(* IEC 61131-3 sources: 2026_Projet_YGO_ExcavatriceDragage/CODE/TESTS, 3 files *)

(* ---- PRG_SafetyValidation.st ---- *)
(* ═══════════════════════════════════════════════════════════════
   🧪 PRG_SafetyValidation — Validateur Automatique de Sécurité (CI/CD)
   ───────────────────────────────────────────────────────────────
   🎯 Rôle : Exécute une suite de scénarios de tests réglementaires
      (NF EN ISO 13849-1) sur le bloc FB_Safety_EmergencyManagement.
   ⚙️ S'exécute uniquement si GVL_Simulation.SimulationModeActive est actif.
   ═══════════════════════════════════════════════════════════════ *)

PROGRAM PRG_SafetyValidation
VAR_OUTPUT
    // Rapport de test (CI/CD)
    TestInProgress             : BOOL;
    TC01_NominalArming_Ok      : BOOL;
    TC02_RedundancyFault_Ok    : BOOL;
    TC03_Lockout_Ok            : BOOL;
    AllTestsPassed             : BOOL;
    TestFailed                 : BOOL;
    FailedTestCase             : INT;         // Numéro du scénario en échec
END_VAR
VAR
    StartTests                 : BOOL;        // Commande de démarrage des tests
    TestSeqStep                : INT := 0;    // Séquenceur de test
    TestTimer                  : TON;         // Timer d'attente d'étapes
    OverrideChainTrue          : BOOL := FALSE; // Force l'entrée boucle d'urgence à TRUE
    OverrideChainFalse         : BOOL := FALSE; // Force l'entrée boucle d'urgence à FALSE
    OverrideContactorFalse     : BOOL := FALSE; // Force l'entrée contacteur à FALSE

    // Signaux locaux pour stimuler le bloc sous test
    ArmRequest                 : BOOL;
    ResetFaults                : BOOL;
    CmdEmergencyCutOff         : BOOL;
END_VAR

// === IMPLEMENTATION ===

// ⛔ Neutralisation si la simulation globale n'est pas active (sécurité physique)
IF NOT GVL_Simulation.SimulationModeActive THEN
    TestSeqStep := 0;
    TestInProgress := FALSE;
    RETURN;
END_IF;

// ⏱️ Timer général d'étape
TestTimer(IN := (TestSeqStep <> 0), PT := T#10s);

// 🔀 Séquenceur de Test Automatique
CASE TestSeqStep OF

    0: // IDLE — En attente du départ de test
        IF StartTests THEN
            StartTests := FALSE;
            TestInProgress := TRUE;
            TC01_NominalArming_Ok := FALSE;
            TC02_RedundancyFault_Ok := FALSE;
            TC03_Lockout_Ok := FALSE;
            AllTestsPassed := FALSE;
            TestFailed := FALSE;
            FailedTestCase := 0;
            OverrideChainTrue := FALSE;
            OverrideChainFalse := FALSE;
            OverrideContactorFalse := FALSE;
            TestSeqStep := 10;
        END_IF;

    // ─────────────────────────────────────────────────────────────────
    // 🧪 SCÉNARIO 1 : Séquence Nominale (TC-01)
    // ─────────────────────────────────────────────────────────────────
    10: // Phase 1.1 : Initialisation saine
        ResetFaults := TRUE;
        IF NOT PRG_10_Outputs.instSafetyEmergencyManagement.RedundancyTestFailed AND
           NOT PRG_10_Outputs.instSafetyEmergencyManagement.EmergencyArmingFailed THEN
            ResetFaults := FALSE;
            TestSeqStep := 11;
        END_IF;

    11: // Phase 1.2 : Envoi demande réarmement
        ArmRequest := TRUE;
        TestSeqStep := 12;

    12: // Phase 1.3 : Vérification début d'auto-test
        ArmRequest := FALSE;
        IF PRG_10_Outputs.instSafetyEmergencyManagement.ArmingSeqStep = 1 THEN
            TestSeqStep := 13;
        END_IF;

    13: // Phase 1.4 : Attente réussite de l'auto-test et début impulsion armement
        IF PRG_10_Outputs.instSafetyEmergencyManagement.ArmingSeqStep = 5 THEN
            TestSeqStep := 14;
        END_IF;

    14: // Phase 1.5 : Attente fin de l'impulsion et confirmation armement
        IF PRG_00_Inputs.EmergencyStopOk AND PRG_10_Outputs.instSafetyEmergencyManagement.ArmingSeqStep = 0 THEN
            // Armé nominalement ! Maintenant on teste le Trip d'urgence
            TestSeqStep := 15;
        END_IF;

    15: // Phase 1.6 : Simulation d'un appui bouton d'urgence (Coupure franche)
        OverrideChainFalse := TRUE;
        TestSeqStep := 16;

    16: // Phase 1.7 : Vérification coupure instantanée
        IF NOT PRG_10_Outputs.PowerCutOff_A_RQ AND NOT PRG_10_Outputs.PowerCutOff_B_RQ AND NOT PRG_00_Inputs.EmergencyStopOk THEN
            // Coupure validée, on relâche le bouton d'urgence (doit rester coupé)
            OverrideChainFalse := FALSE;
            TestSeqStep := 17;
        END_IF;

    17: // Phase 1.8 : Vérification de l'auto-maintien (Latch)
        IF NOT PRG_10_Outputs.PowerCutOff_A_RQ AND NOT PRG_10_Outputs.PowerCutOff_B_RQ THEN
            TC01_NominalArming_Ok := TRUE;
            TestSeqStep := 20; // Passer au test de redondance
        ELSE
            TestFailed := TRUE;
            FailedTestCase := 1;
            TestSeqStep := 999;
        END_IF;

    // ─────────────────────────────────────────────────────────────────
    // 🧪 SCÉNARIO 2 : Défaut de Redondance (TC-02)
    // ─────────────────────────────────────────────────────────────────
    20: // Phase 2.1 : Acquitter le défaut précédent et relancer l'armement
        ResetFaults := TRUE;
        IF NOT PRG_10_Outputs.instSafetyEmergencyManagement.RedundancyTestFailed THEN
            ResetFaults := FALSE;
            ArmRequest := TRUE;
            TestSeqStep := 21;
        END_IF;

    21: // Phase 2.2 : Attente de l'auto-test canal A
        ArmRequest := FALSE;
        IF PRG_10_Outputs.instSafetyEmergencyManagement.ArmingSeqStep = 1 THEN
            // Simuler contacteur A soudé : la chaîne d'urgence reste fermée (TRUE)
            // malgré l'ordre de coupure du canal A.
            OverrideChainTrue := TRUE;
            TestSeqStep := 22;
        END_IF;

    22: // Phase 2.3 : Vérification de la détection du défaut (dans les 200ms)
        IF PRG_10_Outputs.instSafetyEmergencyManagement.RedundancyTestFailed AND
           PRG_10_Outputs.instSafetyEmergencyManagement.ArmingSeqStep = 0 THEN
            // Détection réussie ! Les sorties doivent être inhibées.
            OverrideChainTrue := FALSE;
            TC02_RedundancyFault_Ok := TRUE;
            TestSeqStep := 30; // Passer au test de Lockout
        ELSIF TestTimer.Q THEN
            // Timeout -> Échec du test de redondance
            OverrideChainTrue := FALSE;
            TestFailed := TRUE;
            FailedTestCase := 2;
            TestSeqStep := 999;
        END_IF;

    // ─────────────────────────────────────────────────────────────────
    // 🧪 SCÉNARIO 3 : Verrouillage temporel (TC-03)
    // ─────────────────────────────────────────────────────────────────
    30: // Phase 3.1 : Acquitter et lancer un armement condamné à échouer
        ResetFaults := TRUE;
        IF NOT PRG_10_Outputs.instSafetyEmergencyManagement.RedundancyTestFailed THEN
            ResetFaults := FALSE;
            ArmRequest := TRUE;
            // Bloquer le contacteur de puissance à FALSE
            OverrideContactorFalse := TRUE;
            TestSeqStep := 31;
        END_IF;

    31: // Phase 3.2 : Attente de l'échec de confirmation d'armement (Step 6 -> Lockout)
        ArmRequest := FALSE;
        IF PRG_10_Outputs.instSafetyEmergencyManagement.EmergencyArmingFailed AND
           PRG_10_Outputs.instSafetyEmergencyManagement.EmergencyArmingLockoutActive THEN
            TestSeqStep := 32;
        END_IF;

    32: // Phase 3.3 : Tenter de réarmer immédiatement pendant le lockout de 5s
        ArmRequest := TRUE;
        TestSeqStep := 33;

    33: // Phase 3.4 : Vérifier que la demande de réarmement est ignorée
        ArmRequest := FALSE;
        IF PRG_10_Outputs.instSafetyEmergencyManagement.ArmingSeqStep <> 0 THEN
            // Pas normal, on a démarré pendant le lockout !
            OverrideContactorFalse := FALSE;
            TestFailed := TRUE;
            FailedTestCase := 3;
            TestSeqStep := 999;
        ELSE
            // Demande ignorée avec succès, on attend la fin du lockout
            TestSeqStep := 34;
        END_IF;

    34: // Phase 3.5 : Attente de la libération du verrouillage (5s)
        IF NOT PRG_10_Outputs.instSafetyEmergencyManagement.EmergencyArmingLockoutActive THEN
            // Lockout terminé, on désactive le blocage contacteur
            OverrideContactorFalse := FALSE;
            ResetFaults := TRUE;
            TestSeqStep := 35;
        END_IF;

    35: // Phase 3.6 : Valider qu'un réarmement normal est à nouveau possible
        ResetFaults := FALSE;
        ArmRequest := TRUE;
        TestSeqStep := 36;

    36: // Phase 3.7 : Confirmation finale de l'armement après lockout
        ArmRequest := FALSE;
        IF PRG_00_Inputs.EmergencyStopOk THEN
            TC03_Lockout_Ok := TRUE;
            AllTestsPassed := TRUE;
            TestSeqStep := 100; // Succès global !
        ELSIF TestTimer.Q THEN
            TestFailed := TRUE;
            FailedTestCase := 4;
            TestSeqStep := 999;
        END_IF;

    100: // SUCCÈS GLOBAL
        TestInProgress := FALSE;
        TestSeqStep := 0;

    999: // ÉCHEC
        TestInProgress := FALSE;
        TestSeqStep := 0;

END_CASE;

// === SURCHARGE DES SIGNALS DE SIMULATION (OVERRIDE INTERNE) ===
// Puisque PRG_SafetyValidation tourne APRÈS PRG_00_Inputs, nous surchargeons les
// variables d'entrées physiques pour injecter nos défauts de tests contrôlés.

IF OverrideChainTrue THEN
    PRG_00_Inputs.EmergencyChain := TRUE;
END_IF;

IF OverrideChainFalse THEN
    PRG_00_Inputs.EmergencyChain := FALSE;
END_IF;

IF OverrideContactorFalse THEN
    PRG_00_Inputs.EmergencyStopOk := FALSE;
END_IF;

(* ---- PRG_Test_FinalBrakePowerInterlock.st ---- *)
(* ═══════════════════════════════════════════════════════════════
   🧪 PRG_Test_FinalBrakePowerInterlock — Tests PLC préparés Lot 3A
   ───────────────────────────────────────────────────────────────
   ⚠️ Non exécuté : appeler uniquement dans un projet de test CODESYS.
   ⏱️ Les temporisations sont celles réelles des FB. Les résultats restent
      des preuves préparées, pas une exécution CODESYS déclarée.
   🏗️ Précondition statique : les instances production sont exclusivement dans
      PRG_10_Outputs_LD ; ce test unitaire compose les FB directement.
   ═══════════════════════════════════════════════════════════════ *)
PROGRAM PRG_Test_FinalBrakePowerInterlock
VAR
    InterlockM1 : FB_WinchOutputInterlock_LD;
    InterlockM2 : FB_WinchOutputInterlock_LD;
    InterlockM3 : FB_TranslationOutputInterlock_LD;
    ScenarioStep : INT;
    ResetRequest : BOOL;
    EnableRequest : BOOL := TRUE;
    EmergencyStopOkRequest : BOOL := TRUE;
    SafeStopRequest : BOOL;
    BrakeConfirmed : BOOL;
    ContactorsReleased : BOOL;
    RequestedStepM1 : INT;
    RequestedStepM2 : INT;
    RequestedContactorM1_1 : BOOL;
    RequestedContactorM1_2 : BOOL;
    RequestedContactorM1_3 : BOOL;
    RequestedContactorM1_4 : BOOL;
    RequestedContactorM2_1 : BOOL;
    RequestedContactorM2_2 : BOOL;
    RequestedContactorM2_3 : BOOL;
    RequestedContactorM2_4 : BOOL;
    M2TableMappingPreservedOk : BOOL;
    RequestedDriveControlWord : WORD := 0;
    ScenarioDone : BOOL;
    ScenarioFailed : BOOL;

    M1BrakeTimeoutOk : BOOL;
    M1EnableLatchHeldOk : BOOL;
    M1EmergencyStopLatchHeldOk : BOOL;
    M1EnableRecoveryOk : BOOL;
    M1EmergencyStopRecoveryOk : BOOL;
    M1ResetOk : BOOL;
    M1StepProgressionOk : BOOL := TRUE;
    M1TransitionViolation : BOOL;
    M1PreviousAuthorizedStep : INT;

    M2BrakeTimeoutOk : BOOL;
    M2EnableLatchHeldOk : BOOL;
    M2EmergencyStopLatchHeldOk : BOOL;
    M2FeedbackOffWaitOk : BOOL;
    M2RestartDelayOk : BOOL;
    StopGateOk : BOOL := TRUE;

    M3BrakeGateOk : BOOL;
    M3BrakeTimeoutOk : BOOL;
    M3EnableLatchHeldOk : BOOL;
    M3EmergencyStopLatchHeldOk : BOOL;
    M3ResetWordOk : BOOL;
    M3PostResetHeldOk : BOOL;
    M3RestartAfterNewRequestOk : BOOL;
    M3EnableGateOk : BOOL;
    M3EmergencyStopGateOk : BOOL;
    M3SafeStopRampOk : BOOL;

    // Test end-to-end FB_Winch : la temporisation métier T#1s500ms reste
    // distincte du filet final T#1s250ms de FB_WinchOutputInterlock_LD.
    WinchBusiness : FB_Winch;
    WinchBusinessTable : ST_SpeedStepTable;
    WinchBusinessPreviousStep : INT;
    WinchBusinessTransitionViolation : BOOL;
    WinchBusinessDelayObserved : BOOL;
    WinchBusinessTestPassed : BOOL;

    // Chaîne réelle M3 : FB_Translation produit la rampe, puis l'interlock _LD
    // applique la frontière finale. Ce scénario n'injecte jamais une fréquence.
    TranslationIntegration : FB_Translation;
    TranslationIntegrationInterlock : FB_TranslationOutputInterlock_LD;
    TranslationIntegrationSafeStop : BOOL;
    TranslationIntegrationInitialFreqHz : REAL;
    TranslationIntegrationRampObservedOk : BOOL;
    TranslationIntegrationFinalFollowOk : BOOL;
END_VAR

// ── FB_Winch : temporisation métier réelle T#1s500ms ───────────────────
// Table cumulative minimale valide pour faire atteindre le palier 5 en test.
WinchBusinessTable.P1R1 := FALSE; WinchBusinessTable.P1R2 := FALSE;
WinchBusinessTable.P1R3 := FALSE; WinchBusinessTable.P1R4 := FALSE;
WinchBusinessTable.P2R1 := TRUE;  WinchBusinessTable.P2R2 := FALSE;
WinchBusinessTable.P2R3 := FALSE; WinchBusinessTable.P2R4 := FALSE;
WinchBusinessTable.P3R1 := TRUE;  WinchBusinessTable.P3R2 := TRUE;
WinchBusinessTable.P3R3 := FALSE; WinchBusinessTable.P3R4 := FALSE;
WinchBusinessTable.P4R1 := TRUE;  WinchBusinessTable.P4R2 := TRUE;
WinchBusinessTable.P4R3 := TRUE;  WinchBusinessTable.P4R4 := FALSE;
WinchBusinessTable.P5R1 := TRUE;  WinchBusinessTable.P5R2 := TRUE;
WinchBusinessTable.P5R3 := TRUE;  WinchBusinessTable.P5R4 := TRUE;
WinchBusinessTable.StepThreshold_Pct := [10.0, 20.0, 30.0, 40.0, 100.0];
WinchBusiness(
    Enable := TRUE, Reset := FALSE, EmergencyStopOk := TRUE, Mode := E_Mode.MAINT_N1,
    StartStop := TRUE, SafeStop := FALSE, ForbidDescent := FALSE, ForbidAscent := FALSE,
    Direction := 1, SpeedRefPct := 100.0, SpeedStepTable := WinchBusinessTable,
    FwdRevSpeedFeedbackOff := TRUE, BrakeFeedback := FALSE,
    BypassContactorCheck := TRUE, BypassGlobal := FALSE,
    Homed := TRUE, HomingSuspect := FALSE, CablePosM := 0.0
);
IF WinchBusiness.StepNumber <> WinchBusinessPreviousStep THEN
    IF (WinchBusiness.StepNumber <> (WinchBusinessPreviousStep + 1))
       OR (WinchBusiness.BusinessStepDelayElapsed < T#1s500ms) THEN
        WinchBusinessTransitionViolation := TRUE;
    END_IF;
    WinchBusinessPreviousStep := WinchBusiness.StepNumber;
END_IF;
IF (WinchBusiness.RequestedStep > WinchBusiness.StepNumber)
   AND (WinchBusiness.BusinessStepDelayElapsed >= T#1s500ms) THEN
    WinchBusinessDelayObserved := TRUE;
END_IF;
WinchBusinessTestPassed := (WinchBusiness.StepNumber = 5)
                           AND WinchBusinessDelayObserved
                           AND NOT WinchBusinessTransitionViolation;

// Les trois interlocks sont appelés chaque cycle. La machine de scénario
// modifie uniquement les entrées pour rendre les transitions observables.
InterlockM1(
    Enable := EnableRequest,
    Reset := ResetRequest,
    EmergencyStopOk := EmergencyStopOkRequest,
    SafeStop := SafeStopRequest,
    BrakeReleaseRequest := (RequestedStepM1 > 0),
    BrakeCommandOpenConfirmed := BrakeConfirmed,
    FwdRevSpeedFeedbackOff := ContactorsReleased,
    RequestedRelayFwd := TRUE,
    RequestedRelayRev := FALSE,
    RequestedContactor1 := RequestedContactorM1_1,
    RequestedContactor2 := RequestedContactorM1_2,
    RequestedContactor3 := RequestedContactorM1_3,
    RequestedContactor4 := RequestedContactorM1_4,
    RequestedStep := RequestedStepM1
);
InterlockM2(
    Enable := EnableRequest,
    Reset := ResetRequest,
    EmergencyStopOk := EmergencyStopOkRequest,
    SafeStop := SafeStopRequest,
    BrakeReleaseRequest := (RequestedStepM2 > 0),
    BrakeCommandOpenConfirmed := BrakeConfirmed,
    FwdRevSpeedFeedbackOff := ContactorsReleased,
    RequestedRelayFwd := TRUE,
    RequestedRelayRev := FALSE,
    RequestedContactor1 := RequestedContactorM2_1,
    RequestedContactor2 := RequestedContactorM2_2,
    RequestedContactor3 := RequestedContactorM2_3,
    RequestedContactor4 := RequestedContactorM2_4,
    RequestedStep := RequestedStepM2
);
// Le mapping contacteurs reste celui produit par FB_Winch. Cas volontairement
// non cumulatif M2 : seul R4 est demandé au palier 2 (ex. table Benne dynamique).
// L'interlock doit le transmettre à l'identique dès que le palier est autorisé.

InterlockM3(
    Enable := EnableRequest,
    Reset := ResetRequest,
    EmergencyStopOk := EmergencyStopOkRequest,
    SafeStop := SafeStopRequest,
    BrakeReleaseRequest := (RequestedDriveControlWord = 1) OR (RequestedDriveControlWord = 2),
    BrakeCommandOpenConfirmed := BrakeConfirmed,
    // IEC SEL(G, IN0, IN1) : G=FALSE → demande normale (1), G=TRUE → reset AC600 (7).
    RequestedDriveControlWord := SEL((ScenarioStep = 95) OR (ScenarioStep = 96), RequestedDriveControlWord, 7),
    RequestedDriveFreqHz := 20.0
);

// Intégration réelle M3 : production par FB_Translation, puis filtre final _LD.
TranslationIntegration(
    Enable := TRUE, Reset := FALSE, EmergencyStopOk := TRUE, Mode := E_Mode.MAINT_N1,
    StartStop := (ScenarioStep >= 110) AND (ScenarioStep < 130),
    SafeStop := TranslationIntegrationSafeStop, Direction := 1, SpeedRefPct := 50.0,
    PositionSensorTarget := FALSE, SlowdownSensor := FALSE,
    LimitSwitchFwd := FALSE, LimitSwitchRev := FALSE,
    DriveStatusWord := 16#0000, DriveActualFreqHz := 0.0,
    BypassContactorCheck := TRUE, BypassLimitSwitch := FALSE, BrakeFeedback := FALSE,
    CfgRampAccelRate := 100.0, CfgRampDecelNormalRate := 100.0, CfgRampDecelFastRate := 1000.0,
    DriveFreqScaleMaxHz := 60.0
);
TranslationIntegrationInterlock(
    Enable := TRUE, Reset := FALSE, EmergencyStopOk := TRUE,
    SafeStop := TranslationIntegrationSafeStop,
    BrakeReleaseRequest := TranslationIntegration.BrakeReleaseRequest,
    BrakeCommandOpenConfirmed := TranslationIntegration.BrakeReleaseRequest,
    RequestedDriveControlWord := TranslationIntegration.RequestedDriveControlWord,
    RequestedDriveFreqHz := TranslationIntegration.RequestedDriveFreqHz
);

// Chaque hausse M1 doit être adjacente et ne peut apparaître qu'après T#1s250ms.
// StepDelayElapsed est capturé par l'interlock au scan exact de la transition.
IF (RequestedStepM1 = 5) AND (InterlockM1.AuthorizedStep <> M1PreviousAuthorizedStep) THEN
    IF (InterlockM1.AuthorizedStep <> (M1PreviousAuthorizedStep + 1))
       OR (InterlockM1.StepDelayElapsed < T#1s250ms) THEN
        M1TransitionViolation := TRUE;
    END_IF;
    M1PreviousAuthorizedStep := InterlockM1.AuthorizedStep;
END_IF;

ResetRequest := FALSE;
CASE ScenarioStep OF
    0: // Initialisation : frein serré, retours contacteurs retombés.
        BrakeConfirmed := FALSE;
        ContactorsReleased := TRUE;
        RequestedStepM1 := 0;
        RequestedStepM2 := 0;
        RequestedContactorM1_1 := FALSE; RequestedContactorM1_2 := FALSE;
        RequestedContactorM1_3 := FALSE; RequestedContactorM1_4 := FALSE;
        RequestedContactorM2_1 := FALSE; RequestedContactorM2_2 := FALSE;
        RequestedContactorM2_3 := FALSE; RequestedContactorM2_4 := FALSE;
        RequestedDriveControlWord := 0;
        ScenarioStep := 10;

    10: // M1/M2 : absence confirmation >500ms → défauts mémorisés, puissance nulle.
        RequestedStepM1 := 1;
        RequestedStepM2 := 1;
        RequestedContactorM1_1 := FALSE; // Palier 1 sans contacteur : table métier valide.
        RequestedContactorM2_1 := FALSE; RequestedContactorM2_2 := FALSE;
        RequestedContactorM2_3 := FALSE; RequestedContactorM2_4 := FALSE;
        IF InterlockM1.Error AND InterlockM2.Error THEN
            M1BrakeTimeoutOk := NOT InterlockM1.BrakeCmd AND (InterlockM1.AuthorizedStep = 0);
            M2BrakeTimeoutOk := NOT InterlockM2.BrakeCmd AND (InterlockM2.AuthorizedStep = 0);
            // Cas 1 : Enable retombe PENDANT les deux latch timeout.
            EnableRequest := FALSE;
            ScenarioStep := 11;
        END_IF;

    11: // Les deux latch timeout survivent à Enable=FALSE ; sorties strictement nulles.
        M1EnableLatchHeldOk := InterlockM1.Error AND InterlockM1.RestartInhibit
                               AND NOT InterlockM1.BrakeCmd AND (InterlockM1.AuthorizedStep = 0);
        M2EnableLatchHeldOk := InterlockM2.Error AND InterlockM2.RestartInhibit
                               AND NOT InterlockM2.BrakeCmd AND (InterlockM2.AuthorizedStep = 0);
        EnableRequest := TRUE;
        EmergencyStopOkRequest := FALSE;
        ScenarioStep := 12;

    12: // Cas 2 séparé : les deux latch timeout survivent à EmergencyStopOk=FALSE.
        M1EmergencyStopLatchHeldOk := InterlockM1.Error AND InterlockM1.RestartInhibit
                                      AND NOT InterlockM1.BrakeCmd AND (InterlockM1.AuthorizedStep = 0);
        M2EmergencyStopLatchHeldOk := InterlockM2.Error AND InterlockM2.RestartInhibit
                                      AND NOT InterlockM2.BrakeCmd AND (InterlockM2.AuthorizedStep = 0);
        EmergencyStopOkRequest := TRUE;
        BrakeConfirmed := TRUE; // Cause disparue seulement après les deux gates.
        RequestedStepM1 := 0;
        RequestedStepM2 := 0;
        ScenarioStep := 20;

    20: // Front Reset conscient M1 après disparition de cause.
        ResetRequest := TRUE;
        ScenarioStep := 21;
    21: // Demande zéro obligatoire après Reset, puis vérification interlock toujours inhibé.
        M1ResetOk := NOT InterlockM1.Error;
        RequestedStepM1 := 0;
        M1EnableRecoveryOk := InterlockM1.RestartInhibit AND NOT InterlockM1.BrakeCmd;
        M1PreviousAuthorizedStep := InterlockM1.AuthorizedStep;
        ScenarioStep := 22;
    22: // Nouvelle demande distincte : Enable rétabli, retombée + T#900ms recommencent.
        RequestedStepM1 := 5;
        M1EmergencyStopRecoveryOk := InterlockM1.RestartInhibit OR (InterlockM1.AuthorizedStep = 0);
        ScenarioStep := 30;

    30: // M1 : capture chaque transition 0→1→2→3→4→5.
        IF InterlockM1.AuthorizedStep = 5 THEN
            M1StepProgressionOk := NOT M1TransitionViolation;
            RequestedStepM1 := 0;
            ContactorsReleased := FALSE;
            ScenarioStep := 40;
        END_IF;

    40: // M2 : retour NON retombé → attente explicite, aucun redémarrage.
        RequestedStepM2 := 2;
        // Cas table spécifique M2 : P2 = R4 seul, non cumulatif.
        RequestedContactorM2_1 := FALSE; RequestedContactorM2_2 := FALSE;
        RequestedContactorM2_3 := FALSE; RequestedContactorM2_4 := TRUE;
        M2FeedbackOffWaitOk := (InterlockM2.AuthorizedStep = 0)
                                AND NOT ContactorsReleased;
        ContactorsReleased := TRUE;
        ScenarioStep := 50;

    50: // M2 : après retour retombé, l'autorisation ne vient qu'après T#900ms.
        IF InterlockM2.AuthorizedStep = 2 THEN
            M2RestartDelayOk := M2FeedbackOffWaitOk
                                 AND (InterlockM2.RestartDelayElapsed >= T#900ms);
            M2TableMappingPreservedOk := NOT InterlockM2.Contactor1
                                         AND NOT InterlockM2.Contactor2
                                         AND NOT InterlockM2.Contactor3
                                         AND InterlockM2.Contactor4;
            RequestedStepM2 := 0;
            RequestedContactorM2_4 := FALSE;
            ScenarioStep := 60;
        END_IF;

    60: // Enable coupe immédiatement puissance/frein.
        EnableRequest := FALSE;
        ScenarioStep := 61;
    61:
        StopGateOk := StopGateOk AND NOT InterlockM1.BrakeCmd AND NOT InterlockM2.BrakeCmd
                      AND (InterlockM1.AuthorizedStep = 0) AND (InterlockM2.AuthorizedStep = 0);
        EnableRequest := TRUE;
        EmergencyStopOkRequest := FALSE;
        ScenarioStep := 62;
    62: // EmergencyStopOk coupe immédiatement puissance/frein.
        StopGateOk := StopGateOk AND NOT InterlockM1.BrakeCmd AND NOT InterlockM2.BrakeCmd
                      AND (InterlockM1.AuthorizedStep = 0) AND (InterlockM2.AuthorizedStep = 0);
        EmergencyStopOkRequest := TRUE;
        SafeStopRequest := TRUE;
        ScenarioStep := 63;
    63: // SafeStop ne coupe pas l'interlock : la rampe rapide reste métier.
        // Ici la demande est déjà nulle : les sorties restent donc nulles sans exception _LD.
        StopGateOk := StopGateOk AND (InterlockM1.AuthorizedStep = 0) AND (InterlockM2.AuthorizedStep = 0);
        SafeStopRequest := FALSE;
        BrakeConfirmed := FALSE;
        RequestedDriveControlWord := 1; // Demande normale de marche M3.
        ScenarioStep := 90;

    90: // M3 : aucune fréquence/couple après pré-magnétisation sans confirmation.
        M3BrakeGateOk := (InterlockM3.DriveControlWord = 0) AND (InterlockM3.DriveFreqRefHz = 0.0);
        IF InterlockM3.Error THEN
            M3BrakeTimeoutOk := NOT InterlockM3.BrakeCmd AND InterlockM3.RestartInhibit;
            // Timeout M3 : les deux gates durs suivants ne doivent jamais masquer Error.
            EnableRequest := FALSE;
            ScenarioStep := 91;
        END_IF;

    91: // Timeout M3 persiste pendant Enable=FALSE, sorties sûres.
        M3EnableLatchHeldOk := InterlockM3.Error AND InterlockM3.RestartInhibit
                               AND (InterlockM3.DriveControlWord = 0)
                               AND (InterlockM3.DriveFreqRefHz = 0.0) AND NOT InterlockM3.BrakeCmd;
        EnableRequest := TRUE;
        EmergencyStopOkRequest := FALSE;
        ScenarioStep := 92;

    92: // Timeout M3 persiste pendant EmergencyStopOk=FALSE, sorties sûres.
        M3EmergencyStopLatchHeldOk := InterlockM3.Error AND InterlockM3.RestartInhibit
                                      AND (InterlockM3.DriveControlWord = 0)
                                      AND (InterlockM3.DriveFreqRefHz = 0.0) AND NOT InterlockM3.BrakeCmd;
        EmergencyStopOkRequest := TRUE;
        BrakeConfirmed := TRUE; // Cause disparue après les deux gates.
        ScenarioStep := 95;

    95: // Reset variateur : SEL force word 7, fréquence toujours nulle.
        ResetRequest := TRUE;
        ScenarioStep := 96;
    96:
        M3ResetWordOk := (InterlockM3.DriveControlWord = 7) AND (InterlockM3.DriveFreqRefHz = 0.0);
        RequestedDriveControlWord := 1; // Demande maintenue : doit rester inhibée.
        ScenarioStep := 97;
    97:
        M3PostResetHeldOk := InterlockM3.RestartInhibit
                              AND (InterlockM3.DriveControlWord = 0)
                              AND (InterlockM3.DriveFreqRefHz = 0.0);
        RequestedDriveControlWord := 0; // Neutre explicite obligatoire.
        ScenarioStep := 98;
    98:
        RequestedDriveControlWord := 1; // Nouvelle demande après neutre.
        ScenarioStep := 99;
    99:
        M3RestartAfterNewRequestOk := NOT InterlockM3.RestartInhibit
                                      AND (InterlockM3.DriveControlWord = 1)
                                      AND (InterlockM3.DriveFreqRefHz > 0.0);
        EnableRequest := FALSE;
        ScenarioStep := 100;
    100: // M3 Enable=FALSE : mot, fréquence et frein en position sûre.
        M3EnableGateOk := (InterlockM3.DriveControlWord = 0)
                           AND (InterlockM3.DriveFreqRefHz = 0.0)
                           AND NOT InterlockM3.BrakeCmd;
        EnableRequest := TRUE;
        EmergencyStopOkRequest := FALSE;
        ScenarioStep := 101;
    101: // M3 EmergencyStopOk=FALSE : mot, fréquence et frein en position sûre.
        M3EmergencyStopGateOk := (InterlockM3.DriveControlWord = 0)
                                  AND (InterlockM3.DriveFreqRefHz = 0.0)
                                  AND NOT InterlockM3.BrakeCmd;
        EmergencyStopOkRequest := TRUE;
        ScenarioStep := 110;

    110: // FB_Translation réel : attendre une fréquence amont et finale non nulles.
        IF TranslationIntegrationInterlock.DriveFreqRefHz > 0.0 THEN
            TranslationIntegrationInitialFreqHz := TranslationIntegrationInterlock.DriveFreqRefHz;
            TranslationIntegrationSafeStop := TRUE;
            ScenarioStep := 111;
        END_IF;
    111: // SafeStop : la rampe rapide est produite amont, la frontière _LD la suit.
        IF (TranslationIntegration.RequestedDriveFreqHz > 0.0)
           AND (TranslationIntegration.RequestedDriveFreqHz < TranslationIntegrationInitialFreqHz)
           AND (TranslationIntegrationInterlock.DriveFreqRefHz = TranslationIntegration.RequestedDriveFreqHz)
           AND ((TranslationIntegrationInterlock.DriveControlWord = 1)
                OR (TranslationIntegrationInterlock.DriveControlWord = 0)) THEN
            TranslationIntegrationRampObservedOk := TRUE;
        END_IF;
        IF TranslationIntegration.RequestedDriveFreqHz = 0.0 THEN
            TranslationIntegrationFinalFollowOk := (TranslationIntegrationInterlock.DriveControlWord = 0)
                                                   AND (TranslationIntegrationInterlock.DriveFreqRefHz = 0.0);
            TranslationIntegrationSafeStop := FALSE;
            ScenarioStep := 120;
        END_IF;
    120: // La durée du test métier dépend des TON réels : attendre le palier 5.
        IF WinchBusinessTestPassed THEN
            ScenarioDone := M1BrakeTimeoutOk AND M1ResetOk AND M1StepProgressionOk
                            AND M1EnableLatchHeldOk AND M1EmergencyStopLatchHeldOk
                            AND M1EnableRecoveryOk AND M1EmergencyStopRecoveryOk
                            AND M2BrakeTimeoutOk AND M2EnableLatchHeldOk AND M2EmergencyStopLatchHeldOk
                            AND M2FeedbackOffWaitOk AND M2RestartDelayOk AND M2TableMappingPreservedOk AND StopGateOk
                            AND M3BrakeGateOk AND M3BrakeTimeoutOk
                            AND M3EnableLatchHeldOk AND M3EmergencyStopLatchHeldOk AND M3ResetWordOk
                            AND M3PostResetHeldOk AND M3RestartAfterNewRequestOk
                            AND M3EnableGateOk AND M3EmergencyStopGateOk
                            AND TranslationIntegrationRampObservedOk AND TranslationIntegrationFinalFollowOk
                            AND WinchBusinessTestPassed;
            ScenarioFailed := NOT ScenarioDone;
        END_IF;
ELSE
    ScenarioFailed := TRUE;
END_CASE

(* ---- PRG_Test_KoboldMaintenance.st ---- *)
(* ═══════════════════════════════════════════════════════════════
   🧪 PRG_Test_KoboldMaintenance — Tests PLC isolés T81/T82
   ───────────────────────────────────────────────────────────────
   📄 Doc : DOC/AF_Partie-04_Mode_SemiAuto_Sequenceur_v2.0.md §3ter
   ⚠️ Programme de qualification MANUELLE : non appelé par MainTask.
      L'opérateur l'appelle temporairement dans une tâche de test, pose TestEnable,
      puis lit Passed/Failed. Aucun accès E/S, aucun ordre machine.
   ═══════════════════════════════════════════════════════════════ *)
PROGRAM PRG_Test_KoboldMaintenance
VAR_INPUT
    TestEnable : BOOL;
    ResetTests : BOOL;
END_VAR
VAR_OUTPUT
    Busy       : BOOL;
    Passed     : BOOL;
    Failed     : BOOL;
    ErrorId    : WORD; (* bit0 Dive valide, bit1 Dive invalide, bit2 Extraction, bit3 défaut extraction *)
END_VAR
VAR
    ResetEdge        : R_TRIG;
    DiveValid        : FB_DiveSearch;
    DiveInvalid      : FB_DiveSearch;
    ExtractionValid  : FB_ExtractionSequence;
    ExtractionInvalid: FB_ExtractionSequence;
    DiveValidStep    : INT;
    DiveInvalidStep  : INT;
    ExtractionStep   : INT;
    DiveKobold       : BOOL;
    DiveMotion       : BOOL;
    DivePosition_M   : REAL;
    InvalidKobold    : BOOL;
    InvalidMotion    : BOOL;
    InvalidPosition_M: REAL;
    ExtractionMotion : BOOL;
    ExtractionClosed : BOOL;
    ExtractionBusy   : BOOL;
    ExtractionPos_M  : REAL;
END_VAR

ResetEdge(CLK := ResetTests);
IF ResetEdge.Q OR NOT TestEnable THEN
    Busy := FALSE; Passed := FALSE; Failed := FALSE; ErrorId := 16#0000;
    DiveValidStep := 0; DiveInvalidStep := 0; ExtractionStep := 0;
    DiveKobold := FALSE; DiveMotion := FALSE; DivePosition_M := 1.0;
    InvalidKobold := FALSE; InvalidMotion := FALSE; InvalidPosition_M := 1.0;
    ExtractionMotion := FALSE; ExtractionClosed := FALSE; ExtractionBusy := FALSE; ExtractionPos_M := 0.0;
ELSE
    Busy := NOT Passed AND NOT Failed;

    (* TC-KM-01 : Kobold hors eau 0 → immersion 1 dans fenêtre → fond 0. *)
    CASE DiveValidStep OF
        0: DiveMotion := FALSE; DiveKobold := FALSE; DivePosition_M := 1.0; DiveValidStep := 1;
        1: DiveMotion := FALSE; DiveKobold := FALSE; DivePosition_M := 1.0; DiveValidStep := 2;
        2: DiveMotion := TRUE;  DiveKobold := FALSE; DivePosition_M := 0.4; DiveValidStep := 3;
        3: DiveMotion := TRUE;  DiveKobold := TRUE;  DivePosition_M := 0.0; DiveValidStep := 4;
        4: DiveMotion := TRUE;  DiveKobold := TRUE;  DivePosition_M := -0.1; DiveValidStep := 5;
        5: DiveMotion := TRUE;  DiveKobold := FALSE; DivePosition_M := -0.2; DiveValidStep := 6;
    END_CASE;

    (* TC-KM-02 : front immersion hors fenêtre → T82 / ErrorId bit1. *)
    CASE DiveInvalidStep OF
        0: InvalidMotion := FALSE; InvalidKobold := FALSE; InvalidPosition_M := 1.0; DiveInvalidStep := 1;
        1: InvalidMotion := FALSE; InvalidKobold := FALSE; InvalidPosition_M := 1.0; DiveInvalidStep := 2;
        2: InvalidMotion := TRUE;  InvalidKobold := FALSE; InvalidPosition_M := 0.4; DiveInvalidStep := 3;
        3: InvalidMotion := TRUE;  InvalidKobold := TRUE;  InvalidPosition_M := 0.7; DiveInvalidStep := 4;
    END_CASE;

    (* TC-KM-03 : fond → fermeture → palier 1 sur 2 m → montée nominale. *)
    CASE ExtractionStep OF
        0: ExtractionMotion := FALSE; ExtractionClosed := FALSE; ExtractionBusy := FALSE; ExtractionPos_M := 0.0; ExtractionStep := 1;
        1: ExtractionMotion := FALSE; ExtractionStep := 2;
        2: ExtractionMotion := TRUE;  ExtractionStep := 3;
        3: ExtractionMotion := TRUE;  ExtractionClosed := FALSE; ExtractionBusy := TRUE; ExtractionStep := 4;
        4: ExtractionMotion := TRUE;  ExtractionClosed := TRUE;  ExtractionBusy := FALSE; ExtractionPos_M := 0.0; ExtractionStep := 5;
        5: ExtractionMotion := TRUE;  ExtractionPos_M := 0.0; ExtractionStep := 6;
        6: ExtractionMotion := TRUE;  ExtractionPos_M := 2.0; ExtractionStep := 7;
    END_CASE;
END_IF;

DiveValid(
    Enable := TestEnable, Reset := FALSE, EmergencyStopOk := TRUE, Mode := E_Mode.MAINT_N1,
    MotionRequestActive := DiveMotion, MotionDirection := -1, BucketIsOpen := TRUE,
    KoboldImmersed := DiveKobold, M1Position_M := DivePosition_M, M2Position_M := DivePosition_M,
    PositionsValid := TRUE, DiveStartMin_M := 1.0, ImmersionUpper_M := 0.5, ImmersionLower_M := -0.5
);
DiveInvalid(
    Enable := TestEnable, Reset := FALSE, EmergencyStopOk := TRUE, Mode := E_Mode.MAINT_N1,
    MotionRequestActive := InvalidMotion, MotionDirection := -1, BucketIsOpen := TRUE,
    KoboldImmersed := InvalidKobold, M1Position_M := InvalidPosition_M, M2Position_M := InvalidPosition_M,
    PositionsValid := TRUE, DiveStartMin_M := 1.0, ImmersionUpper_M := 0.5, ImmersionLower_M := -0.5
);
ExtractionValid(
    Enable := TestEnable, Reset := FALSE, EmergencyStopOk := TRUE, Mode := E_Mode.MAINT_N1,
    MotionRequestActive := ExtractionMotion, MotionDirection := 1, BottomPositionConfirmed := TRUE,
    BucketIsClosed := ExtractionClosed, BucketBusy := ExtractionBusy, BucketError := FALSE,
    WinchSyncError := FALSE, M1Position_M := ExtractionPos_M, M2Position_M := ExtractionPos_M,
    M1MeasuredSpeedValid := TRUE, M2MeasuredSpeedValid := TRUE, PositionsValid := TRUE,
    ControlAscentDistance_M := 2.0
);
ExtractionInvalid(
    Enable := TestEnable, Reset := FALSE, EmergencyStopOk := TRUE, Mode := E_Mode.MAINT_N1,
    MotionRequestActive := FALSE, MotionDirection := 0, BottomPositionConfirmed := FALSE,
    BucketIsClosed := FALSE, BucketBusy := FALSE, BucketError := FALSE, WinchSyncError := FALSE,
    M1Position_M := 0.0, M2Position_M := 0.0, M1MeasuredSpeedValid := TRUE,
    M2MeasuredSpeedValid := TRUE, PositionsValid := TRUE, ControlAscentDistance_M := 0.0
);

IF DiveValid.BottomTouchConfirmed THEN ErrorId := ErrorId OR 16#0001; END_IF;
IF DiveInvalid.Error AND ((DiveInvalid.ErrorId AND 16#0002) <> 16#0000) THEN ErrorId := ErrorId OR 16#0002; END_IF;
IF (ExtractionValid.ExtractionState = E_ExtractionSequenceState.CONTROL_ASCENT)
   AND ExtractionValid.ForceMinSpeedStep THEN ErrorId := ErrorId OR 16#0004; END_IF;
IF ExtractionValid.ExtractionState = E_ExtractionSequenceState.NOMINAL_ASCENT
   AND ExtractionValid.AscentPermit THEN ErrorId := ErrorId OR 16#0004; END_IF;
IF ExtractionInvalid.Error AND ((ExtractionInvalid.ErrorId AND 16#0008) <> 16#0000) THEN ErrorId := ErrorId OR 16#0008; END_IF;

IF (ErrorId AND 16#000F) = 16#000F THEN
    Passed := TRUE;
    Busy := FALSE;
END_IF;
